// Mitsubishi GX Works2 project: wave   PLC: FX3U/FX3UC

PROGRAM MAIN
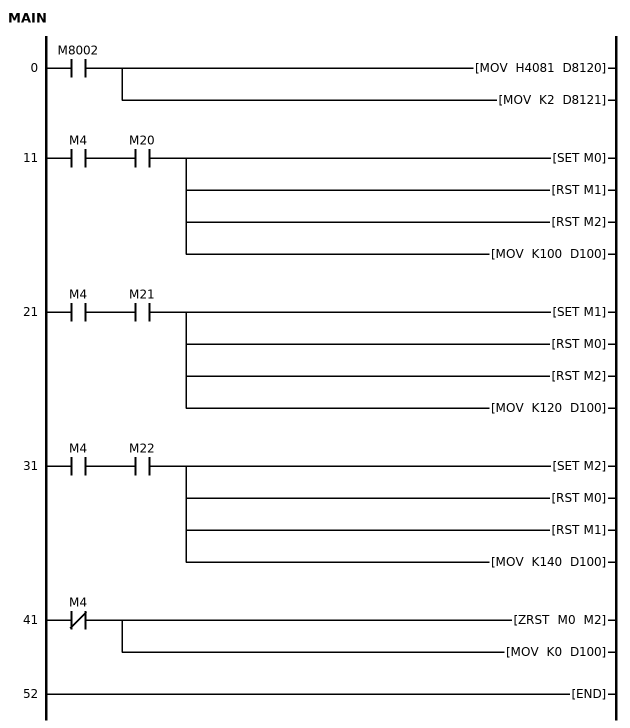
0     LD      M8002
      MOV     H4081 D8120
      MOV     K2 D8121
11    LD      M4
      AND     M20
      SET     M0
      RST     M1
      RST     M2
      MOV     K100 D100
21    LD      M4
      AND     M21
      SET     M1
      RST     M0
      RST     M2
      MOV     K120 D100
31    LD      M4
      AND     M22
      SET     M2
      RST     M0
      RST     M1
      MOV     K140 D100
41    LDI     M4
      ZRST    M0 M2
      MOV     K0 D100
52    END
END_PROGRAM
